TYPE (* A Structure with 8 BOOLS *)
  (* Version 1.0, 2024-02-21, Franz Höpfinger, HR Agrartechnik GmbH *)
  ST08B : STRUCT
    B_00 : BOOL; (* BIT 00 *)
    B_01 : BOOL; (* BIT 01 *)
    B_02 : BOOL; (* BIT 02 *)
    B_03 : BOOL; (* BIT 03 *)
    B_04 : BOOL; (* BIT 04 *)
    B_05 : BOOL; (* BIT 05 *)
    B_06 : BOOL; (* BIT 06 *)
    B_07 : BOOL; (* BIT 07 *)
  END_STRUCT;
END_TYPE
